Fanuc KAREL source: kt00149.KL

-- PROVISIONAL review KL for V770-1; original PC SHA256 431bad141dfbbb8ca2a87a3eef69bcb24ae5698d4beff1f674920280460b8a9b
-- Incomplete behavior may be omitted. Consult companion uncertainty JSON. Do not deploy.
PROGRAM KT00149
%NOLOCKGROUP
VAR
  OUT : INTEGER
-- UNRESOLVED_DECL Y1 type=002018
-- UNRESOLVED_DECL Y2 type=002018
BEGIN
  -- UNRESOLVED_PC offsets 5-19; opcodes 2E,22,9D,33,B2
  -- UNRESOLVED_PC offsets 24-38; opcodes 2E,22,9D,33,B2
  -- UNRESOLVED_PC offsets 43-57; opcodes 2E,22,9D,33,B2
  -- UNRESOLVED_PC offsets 62-76; opcodes 2E,22,9D,33,B2
  -- UNRESOLVED_PC offsets 81-106; opcodes 22,9D,33,B1,22,9D,33,B1,55,23
  -- UNRESOLVED_PC offsets 111-115; opcodes 7F
END KT00149
